Universal Robots PolyScope program: 2exPause.urp

Program 2exPause (installation=default directory=/home/ur/ursim-current/programs createdIn=5.11.8.1010444 lastSavedIn=5.11.8.1010444 robotSerialNumber=20195399999)
Calibrated DH parameters: a=[0, -0.24355, -0.2132, 0, 0, 0]; d=[0.15185, 0, 0, 0.13105, 0.08535, 0.0921]; alpha=[1.570796, 0, 0, 1.570796, -1.570796, 0]; deltaTheta=[0, 0, 0, 0, 0, 0]
BeforeStart
  Script file /home/ur/ursim-current/programs/Script/2_Ex_CountDown_Pause.script
    | def Pause(counter):
    | 	while 0 < counter:
    | 		counter = counter - 1
    | 		sleep(0.001)
    | 	end
    | end
  Pause_in_msec := 1000
Robot Program (runOnlyOnce=false)
  Set DigitalOutput pin=digital_out[0]; digitalValue=1
  Script: Pause(Pause_in_msec)
  Set DigitalOutput pin=digital_out[0]; digitalValue=0
  Script: Pause(Pause_in_msec)
